SUBAPPLICATION ACTION_CLIENT_SEND_GOAL
  (* Standard: 61499-2 *)
  (* Version 1.0, 2023-03-23, Tim Hesse *)
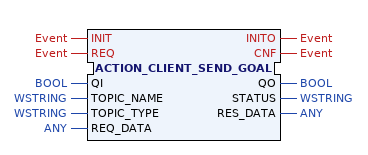
  EVENT_INPUT
    INIT; (* Initialization Request *)
    REQ; (* Normal Execution Request *)
  END_EVENT
  EVENT_OUTPUT
    INITO; (* Initialization Confirm *)
    CNF; (* Execution Confirmation *)
  END_EVENT
  VAR_INPUT
    QI : BOOL; (* Input event qualifier *)
    TOPIC_NAME : WSTRING;
    TOPIC_TYPE : WSTRING;
    REQ_DATA : ANY;
  END_VAR
  VAR_OUTPUT
    QO : BOOL; (* Output event qualifier *)
    STATUS : WSTRING;
    RES_DATA : ANY;
  END_VAR
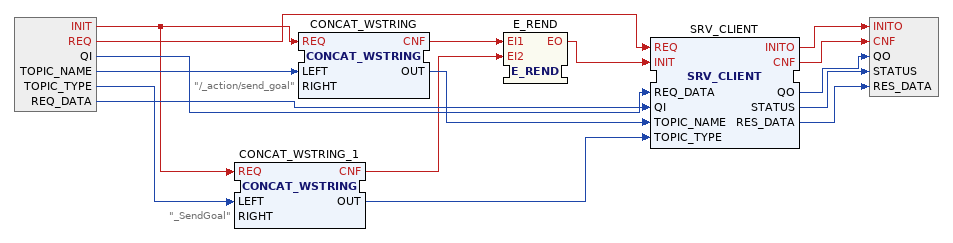
  FBS
    E_REND : E_REND;
  END_FBS
  SUBAPPS
    SRV_CLIENT : SRV_CLIENT;
    CONCAT_WSTRING : CONCAT_WSTRING(RIGHT := "/_action/send_goal");
    CONCAT_WSTRING_1 : CONCAT_WSTRING(RIGHT := "_SendGoal");
  END_SUBAPPS
  EVENT_CONNECTIONS
    SRV_CLIENT.INITO TO INITO;
    SRV_CLIENT.CNF TO CNF;
    REQ TO SRV_CLIENT.REQ;
    CONCAT_WSTRING.CNF TO E_REND.EI1;
    CONCAT_WSTRING_1.CNF TO E_REND.EI2;
    E_REND.EO TO SRV_CLIENT.INIT;
    INIT TO CONCAT_WSTRING.REQ;
    INIT TO CONCAT_WSTRING_1.REQ;
  END_CONNECTIONS
  DATA_CONNECTIONS
    SRV_CLIENT.QO TO QO;
    SRV_CLIENT.STATUS TO STATUS;
    SRV_CLIENT.RES_DATA TO RES_DATA;
    REQ_DATA TO SRV_CLIENT.REQ_DATA;
    QI TO SRV_CLIENT.QI;
    TOPIC_NAME TO CONCAT_WSTRING.LEFT;
    TOPIC_TYPE TO CONCAT_WSTRING_1.LEFT;
    CONCAT_WSTRING.OUT TO SRV_CLIENT.TOPIC_NAME;
    CONCAT_WSTRING_1.OUT TO SRV_CLIENT.TOPIC_TYPE;
  END_CONNECTIONS
END_SUBAPPLICATION
